FUNCTION_BLOCK HRL_ControlOfOutputs
VAR_INPUT
	F4				: BOOL;
	F1				: BOOL;
	A2				: BOOL;
	A1				: BOOL;
	Start			: BOOL;
	CB_forwards 	: BOOL; //GVL_HRL.HRL_MOT_Foerderband_vorwaerts
	CB_backwards 	: BOOL; //GVL_HRL.HRL_MOT_Foerderband_rueckwaerts
	RGB_Forwards01 : BOOL; //GVL_HRL.HRL_MOT_Ausleger_vorwaerts
	RGB_Backwards02 : BOOL; //GVL_HRL.HRL_MOT_Ausleger_vorwaerts
	RGB_Forwards02 : BOOL; //GVL_HRL.HRL_MOT_Ausleger_rueckwaerts
	RGB_Backwards01 : BOOL; //GVL_HRL.HRL_MOT_Ausleger_rueckwaerts
	RGB_VertikalDown01 : BOOL; //GVL_HRL.HRL_MOT_vertikal_runter
	RGB_VertikalUp02 : BOOL; //GVL_HRL.HRL_MOT_vertikal_runter
	RGB_VertikalDown02 : BOOL; //GVL_HRL.HRL_MOT_vertikal_hoch
	RGB_VertikalUp01 : BOOL; //GVL_HRL.HRL_MOT_vertikal_hoch
	RGB_HorizontalForwards01 : BOOL; //GVL_HRL.HRL_MOT_horizontal_zum_Regal
	RGB_HorizontalBackwards02 : BOOL; //GVL_HRL.HRL_MOT_horizontal_zum_Regal
	RGB_HorizontalForwards02 : BOOL; //GVL_HRL.HRL_MOT_horizontal_zum_Foerderband
	RGB_HorizontalBackwards01 : BOOL; //GVL_HRL.HRL_MOT_horizontal_zum_Foerderband
END_VAR
VAR_OUTPUT
	ConveyorBeltForward: BOOL;
	ConveyorBeltBackward: BOOL;
	RGB_Forwards: BOOL;
	RGB_Backwards: BOOL;
	RGB_VerticalDown: BOOL;
	RGB_VerticalUp: BOOL;
	RGB_HorizontalForward: BOOL;
	RGB_HorizontalBackward: BOOL;
	Light_Q1: BOOL;
	Light_Q2: BOOL;
	Light_Q3: BOOL;
END_VAR
VAR
END_VAR

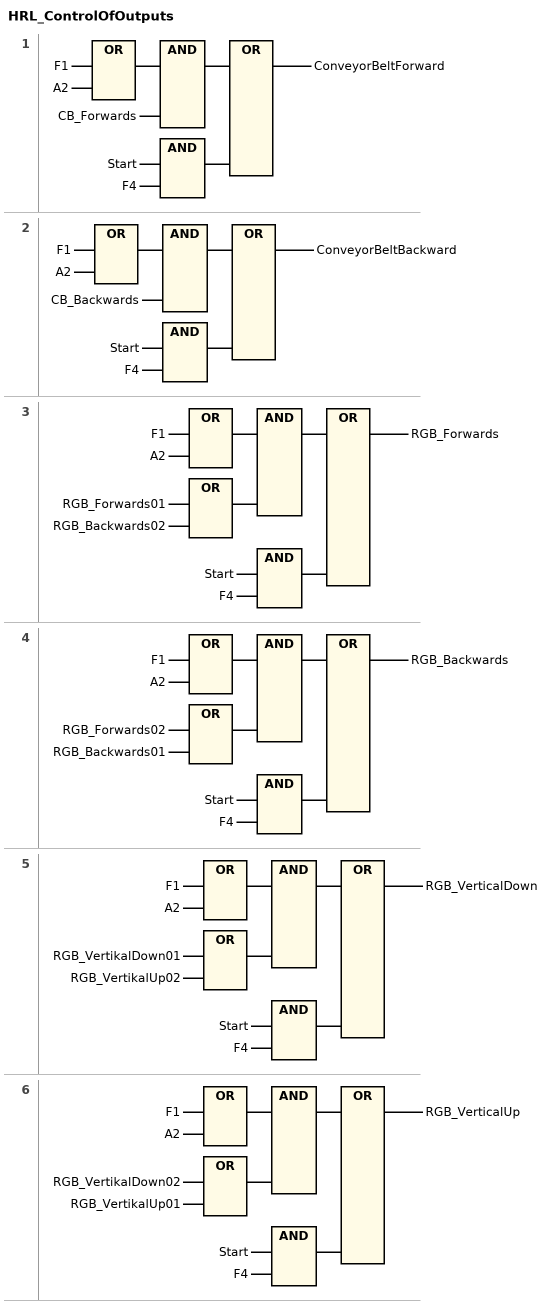
// NETWORK 1
ConveyorBeltForward := (F1 OR A2) AND CB_Forwards OR Start AND F4;

// NETWORK 2
ConveyorBeltBackward := (F1 OR A2) AND CB_Backwards OR Start AND F4;

// NETWORK 3
RGB_Forwards := (F1 OR A2) AND (RGB_Forwards01 OR RGB_Backwards02) OR Start AND F4;

// NETWORK 4
RGB_Backwards := (F1 OR A2) AND (RGB_Forwards02 OR RGB_Backwards01) OR Start AND F4;

// NETWORK 5
RGB_VerticalDown := (F1 OR A2) AND (RGB_VertikalDown01 OR RGB_VertikalUp02) OR Start AND F4;

// NETWORK 6
RGB_VerticalUp := (F1 OR A2) AND (RGB_VertikalDown02 OR RGB_VertikalUp01) OR Start AND F4;

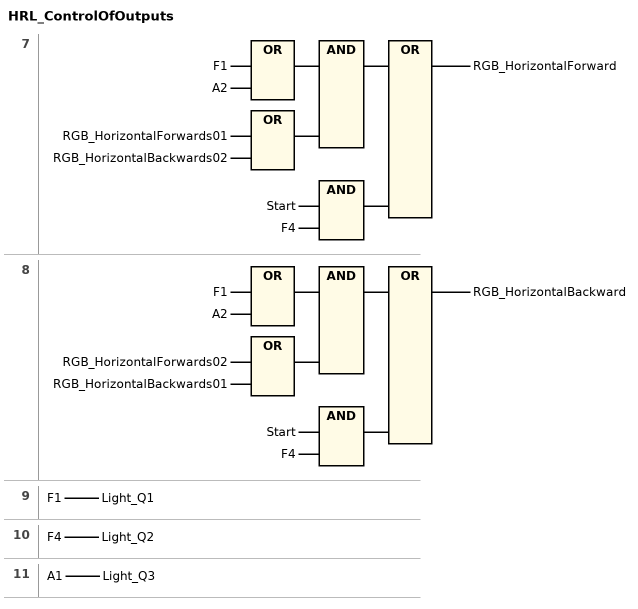
// NETWORK 7
RGB_HorizontalForward := (F1 OR A2) AND (RGB_HorizontalForwards01 OR RGB_HorizontalBackwards02) OR Start AND F4;

// NETWORK 8
RGB_HorizontalBackward := (F1 OR A2) AND (RGB_HorizontalForwards02 OR RGB_HorizontalBackwards01) OR Start AND F4;

// NETWORK 9
Light_Q1 := F1;

// NETWORK 10
Light_Q2 := F4;

// NETWORK 11
Light_Q3 := A1;

END_FUNCTION_BLOCK

(* stored: Version 1.1.0.1, ProductVersion 3.1.4024.15
   POU HRL_ControlOfOutputs: Id {f7623071-88c7-466b-9ed1-985cc415452d}, SpecialFunc None *)
